// TwinCAT 3 PLC project Untitled1
// ProgramVersion: 3.1.4020.5
// libraries:
//   Tc2_Standard, * (Beckhoff Automation GmbH)
//   Tc2_System, * (Beckhoff Automation GmbH)
//   Tc3_Module, * (Beckhoff Automation GmbH)
// project tree:
//   DUTs/ DUT_ENUM_TEST.TcDUT, DUT_STRUCT_TEST.TcDUT
//   / PlcTask.TcTTO
//   POUs/ MAIN.TcPOU
// real-time tasks:
//   TASK PlcTask: cycle T#10ms, priority 20, ADS port 350

CONFIGURATION Untitled1
    RESOURCE PLC ON TwinCAT3
        TASK PlcTask(INTERVAL := T#10ms, PRIORITY := 20);
        PROGRAM MAIN WITH PlcTask : MAIN;
    END_RESOURCE
END_CONFIGURATION

// ---- DUTs/DUT_ENUM_TEST.TcDUT
{attribute 'qualified_only'}
{attribute 'strict'}
TYPE DUT_ENUM_TEST :
(
	zeroeth_member := 0,
	first_member := 1,
	second_member := 2,
	third_member := 3
);
END_TYPE

// ---- DUTs/DUT_STRUCT_TEST.TcDUT
TYPE DUT_STRUCT_TEST :
STRUCT

	{attribute 'pytmc' := '
		pv: ADS_TST:fAmp
		io: o
		pv: ADS_TST:ReadOnly:fAmp
		io: i
	'}
	fAmplitude :	LREAL;
	{attribute 'pytmc' := '
		pv: ADS_TST:FArray
		io: o
		pv: ADS_TST:ReadOnly:FArray
		io: i
	'}
	fArray : ARRAY [1..5] OF LREAL;
	{attribute 'pytmc' := '
		pv: ADS_TST:Str
		io: o
		pv: ADS_TST:ReadOnly:Str
		io: i
	'}
	str	:	STRING(35);


END_STRUCT	
END_TYPE

// ---- POUs/MAIN.TcPOU
PROGRAM MAIN
VAR
	
	{attribute 'pytmc' := '
		pv: ADS_TST:iCycle
		io: io
		pv: ADS_TST:ReadOnly:iCycle
		io: i
	'}
	iCycle : INT;

		{attribute 'pytmc' := '
		pv: ADS_TST:nSignedInt8
		io: io
	'}
	nSignedInt8 : INT;
	
	{attribute 'pytmc' := '
		pv: ADS_TST:diCycle
		io: o
		pv: ADS_TST:ReadOnly:diCycle
		io: i
	'}
	diCycle : DINT;
	
	{attribute 'pytmc' := '
		pv: ADS_TST:bState
		io: o
		pv: ADS_TST:ReadOnly:bState
		io: i
	'}
	bState : BOOL;

	{attribute 'pytmc' := '
		pv: ADS_TST:lrAmp
		io: o
		pv: ADS_TST:ReadOnly:lrAmp
		io: i
	'}
	lrAmplitude :	LREAL;

	{attribute 'pytmc' := '
		pv: ADS_TST:rAmp
		io: o
		pv: ADS_TST:ReadOnly:rAmp
		io: i
	'}
	rAmplitude :	REAL;

	{attribute 'pytmc' := '
		pv: ADS_TST:lrArray
		io: o
		pv: ADS_TST:ReadOnly:lrArray
		io: i
	'}
	lrArray : ARRAY [1..5] OF LREAL;

	{attribute 'pytmc' := '
		pv: ADS_TST:rArray
		io: o
		pv: ADS_TST:ReadOnly:rArray
		io: i
	'}	
	rArray : ARRAY [1..5] OF REAL;

	{attribute 'pytmc' := '
		pv: ADS_TST:iArray
		io: o
		pv: ADS_TST:ReadOnly:iArray
		io: i
	'}
	iArray : ARRAY [1..5] OF INT;

	{attribute 'pytmc' := '
		pv: ADS_TST:diArray
		io: o
		pv: ADS_TST:ReadOnly:rdiArray
		io: i
	'}
	diArray : ARRAY [1..5] OF DINT;
	
	
	{attribute 'pytmc' := '
		pv: ADS_TST:bArray
		io: o
		pv: ADS_TST:ReadOnly:bArray
		io: i
	'}
	bArray : ARRAY [1..5] OF BOOL;
	
	is_true : BOOL;
	is_false : BOOL;
	val : BOOL;
	dval : DINT;

	{attribute 'pytmc' := '
		pv: ADS_TST:Str
		io: o
		pv: ADS_TST:ReadOnly:Str
		io: i
	'}
	sTest	:	STRING(35);
	
	
	
	{attribute 'pytmc' := '
		pv: ADS_TST:eStatus
		io: o
		pv: ADS_TST:ReadOnly:eStatus
		io: i
	'}	
	eStatus	:	DUT_ENUM_TEST;

	{attribute 'pytmc' := '
		pv: ADS_TST:enumArray
		io: o
		pv: ADS_TST:ReadOnly:enumArray
		io: i
	'}	
	enumArray	: ARRAY [1..5] of DUT_ENUM_TEST;

	
	{attribute 'pytmc' := '
		pv: ADS_TST:StrRB
	'}
	//structure_type : DUT_STRUCT_TEST;
	
	// *****************************
	//bool_type : BOOL;
	
	//enum_type : DUT_ENUM_TEST; 
END_VAR

IF bArray[1] = TRUE THEN
	is_true := TRUE;
	is_false := FALSE;

else
	is_true := FALSE;
	is_false := TRUE;
END_IF


val := bArray[1];

END_PROGRAM
